{attribute 'qualified_only'}
{attribute 'strict'}
{attribute 'to_string'}
TYPE
MoverState_e :
(
    OperationDone,     // The operation on the mover is done, a new station needs to be given
    WaitOnNextStation, // wait on the next station to be ready. The waiting depend on the scenario of the next station
    MovingToStation,   // the mover is moving or try to move to the next station
    InStationPos,      // The mover is currently at the station position (aka target pos.), waiting on the process to begin
    InOperation,         // The attached process of the mover is running. The mover is not able to move
    _MAX
);
END_TYPE

(* stored: Version 1.1.0.1, ProductVersion 3.1.4024.6
   EnumerationTextList MoverState_e: Id {10808199-66f7-4ecb-8da3-b56c001df457} *)
